ABB RobotStudio station: Solution2_20220201-115427.rsstn

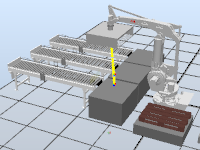
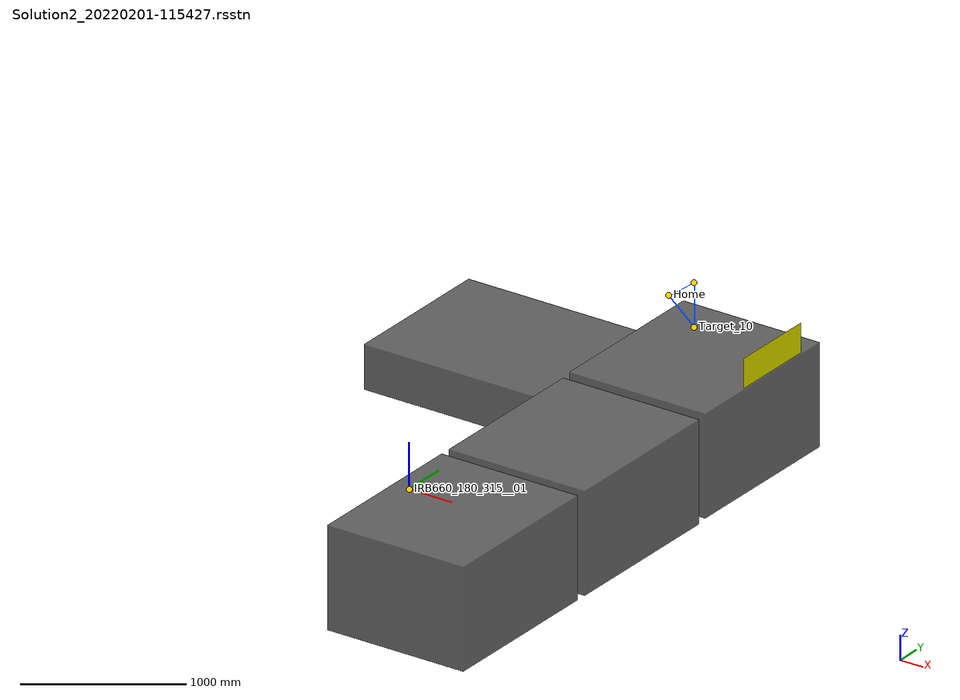
[picture v1: parts stored in the station drawn from their meshes, with robot base, taught points and paths (robot models come from the ABB library and are not in the file)]
Station Solution2 (saved by RobotStudio 21.4.9700.0)
Controller IRB660_180_315
  mechanical unit ROB_1: IRB660_180_315__01, 6 joints, base frame (0, 0, 0) mm
Layout (positions relative to the parent item):
  - IRB660_180_315__01 [mechanism, from Robots\IRB660_180_315__01.rslib] at (0, 0, 0) mm; joint values [0, 0.0198, -0.194, 0] (rad or m)
  - 600_guide [part, from Equipment\Conveyor Guide 600.rslib] at (4720, 275, 0) mm, rotated rx 0 ry 0 rz 180 deg
  - 600_guide_2 [part, from Equipment\Conveyor Guide 600.rslib] at (4720, 1475, 0) mm, rotated rx 0 ry 0 rz 180 deg
  - 600_guide_3 [part, from Equipment\Conveyor Guide 600.rslib] at (4720, -900, 0) mm, rotated rx 0 ry 0 rz 180 deg
  - 1200_4000_h2_2 [part, from Equipment\Conveyor 1200 4000 h2.rslib] at (-1500, -1000, 0) mm, rotated rx 0 ry 0 rz 180 deg
  - 1200_4000_h2_3 [part, from Equipment\Conveyor 1200 4000 h2.rslib] at (-1500, 2000, 0) mm, rotated rx 0 ry 0 rz 180 deg
  - 1200_4000_h2_4 [part, from Equipment\Conveyor 1200 4000 h2.rslib] at (-1500, 500, 0) mm, rotated rx 0 ry 0 rz 180 deg
  - 1200_4800_h2_2 [part, from Equipment\Conveyor 1200 4800 h2.rslib] at (-6865.5, 2181.45, 0) mm, rotated rx 0 ry 0 rz -90 deg
  - Pieza_1 [part] at (-5740.3, -4363.37, 0) mm, rotated rx 0 ry 0 rz 90 deg, size 1600 x 1000 x 355 mm
  - wraping_1 [part] at (-6239.59, -3461.03, 366.67) mm, rotated rx 0 ry 0 rz -90 deg, size 2370 x 1393.7 x 2100 mm
  - wraping_2 [part] at (-6238.99, -3463.39, 358.4) mm, rotated rx 0 ry 0 rz -90 deg, size 1400 x 1393.6 x 350 mm
  - wraping_3 [part] at (-6242.7, -3445.47, -111.4) mm, rotated rx 90 ry 0 rz -90 deg, size 323.7 x 500 x 658.2 mm
  - Pieza_4 [part] at (-1012.61, 969.79, 0) mm, size 1300 x 1100 x 300 mm
  - Pieza_6 [part] at (689.01, 695.64, 0) mm, size 1000 x 1200 x 700 mm
  - Pieza_7 [part] at (702.6, -1863.75, 0) mm, size 1000 x 1200 x 700 mm
  - Pieza_8 [part] at (703.57, -589.74, 0) mm, size 1000 x 1200 x 700 mm
  - Mi_mecanismo [mechanism] at (1910, 0, 2093) mm; joint values [0, 0] (rad or m)
      TCP Mi_mecanismo_1 at (1.05, 425.12, 399.16) mm, rotated rx 90 ry 0 rz 180 deg
      links: L1, L2, L3
  - Euro Pallet [graphiccomponentgroup, from Equipment\Euro Pallet.rslib] at (223.77, 1878.53, 297.19) mm, rotated rx 0 ry 0 rz 180 deg
    - Body 1 [part, from Equipment\Euro Pallet.rslib]
  - Euro Pallet_2 [graphiccomponentgroup, from Equipment\Euro Pallet.rslib] at (-1565.85, 804.31, 434.35) mm, rotated rx 0 ry 0 rz 90 deg
    - Body 1 [part, from Equipment\Euro Pallet.rslib]
  - Pieza_19 [part] at (1001.17, 2703.27, 775) mm, rotated rx 0 ry 0 rz 90 deg, size 425 x 325 x 180 mm
  - Componente inteligente_1 [smart component]
      signals: DI Start, DI Cinta, DI Coger, DI Soltar, DO Sensor1
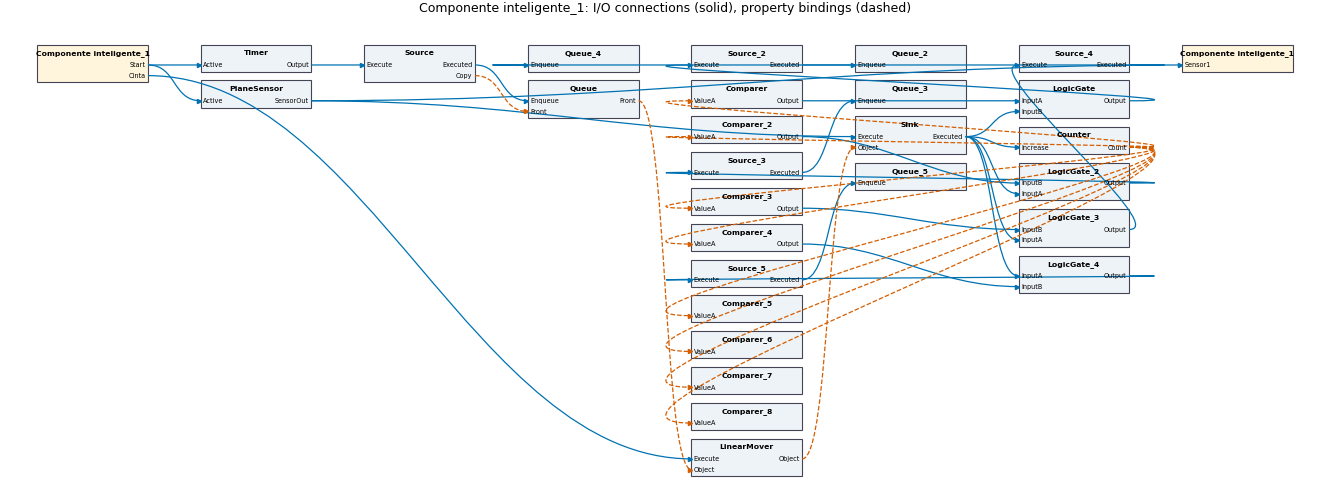
      connections:
        Componente inteligente_1.Start -> Timer.Active
        Timer.Output -> Source.Execute
        Source.Executed -> Queue.Enqueue
        Componente inteligente_1.Cinta -> LinearMover.Execute
        Componente inteligente_1.Start -> PlaneSensor.Active
        PlaneSensor.SensorOut -> Sink.Execute
        Source_2.Executed -> Queue_2.Enqueue
        Sink.Executed -> Counter.Increase
        LogicGate.Output -> Source_2.Execute
        Comparer.Output -> LogicGate.InputA
        Sink.Executed -> LogicGate.InputB
        Comparer_2.Output -> LogicGate_2.InputB
        Sink.Executed -> LogicGate_2.InputA
        LogicGate_2.Output -> Source_3.Execute
        Source_3.Executed -> Queue_3.Enqueue
        PlaneSensor.SensorOut -> Componente inteligente_1.Sensor1
        Comparer_3.Output -> LogicGate_3.InputB
        LogicGate_3.Output -> Source_4.Execute
        Sink.Executed -> LogicGate_3.InputA
        Source_4.Executed -> Queue_4.Enqueue
        Sink.Executed -> LogicGate_4.InputA
        Comparer_4.Output -> LogicGate_4.InputB
        LogicGate_4.Output -> Source_5.Execute
        Source_5.Executed -> Queue_5.Enqueue
        Source.Copy => Queue.Front
        Queue.Front => LinearMover.Object
        LinearMover.Object => Sink.Object
        Counter.Count => Comparer.ValueA
        Counter.Count => Comparer_2.ValueA
        Counter.Count => Comparer_3.ValueA
        Counter.Count => Comparer_4.ValueA
        Counter.Count => Comparer_5.ValueA
        Counter.Count => Comparer_6.ValueA
        Counter.Count => Comparer_7.ValueA
        Counter.Count => Comparer_8.ValueA
    - LinearMover [smart component, from Components\LinearMover.rslib]
        properties: Object=(none); Direction=[-0.001 0 0]; Speed=0.7; Reference=Global; ReferenceObject=(none)
    - PlaneSensor [smart component, from Components\PlaneSensor.rslib] at (1831.92, 892.97, 831.06) mm, rotated rx 0 ry -90 rz 0 deg
        properties: Origin=[0 0 0]; Axis1=[0.2 0 0]; Axis2=[0 0.6 0]; SensedPart=(none)
      - _sensorPart_ [part], size 200 x 600 x 0 mm
    - Attacher [smart component, from Components\Attacher.rslib]
        properties: Parent=(none); Flange=0; Child=(none); Mount=false; Offset=[0 0 0]; Orientation=[0 0 0]
    - Detacher [smart component, from Components\Detacher.rslib]
        properties: Child=(none); KeepPosition=true
    - Queue [smart component, from Components\Queue.rslib]
        properties: Back=(none); Front=(none); Queue=; NumberOfObjects=0
    - Source [smart component, from Components\Source.rslib]
        properties: Source=Pieza_19; Copy=(none); Parent=(none); Position=[4.6 0.975 0.775]; Orientation=[0 0 1.5707963267949]; Transient=true; PhysicsBehavior=0
    - Timer [smart component, from Components\Timer.rslib]
        properties: StartTime=0; Interval=4; Repeat=true; CurrentTime=27.336
    - Sink [smart component, from Components\Sink.rslib]
        properties: Object=(none)
    - Source_2 [smart component, from Components\Source.rslib]
        properties: Source=Pieza_19; Copy=(none); Parent=(none); Position=[1.015 1.47 0.7]; Orientation=[0 0 1.5707963267949]; Transient=false; PhysicsBehavior=0
    - Source_3 [smart component, from Components\Source.rslib]
        properties: Source=Pieza_19; Copy=(none); Parent=(none); Position=[1.345 1.47 0.7]; Orientation=[0 0 1.5707963267949]; Transient=false; PhysicsBehavior=0
    - Source_4 [smart component, from Components\Source.rslib]
        properties: Source=Pieza_19; Copy=(none); Parent=(none); Position=[1.675 1.47 0.7]; Orientation=[0 0 1.5707963267949]; Transient=false; PhysicsBehavior=0
    - Queue_2 [smart component, from Components\Queue.rslib]
        properties: Back=(none); Front=(none); Queue=; NumberOfObjects=0
    - Counter [smart component, from Components\Counter.rslib]
        properties: Count=5
    - LogicGate [smart component, from Components\LogicGate.rslib]
        properties: Operator=AND; Delay=0
    - Comparer [smart component, from Components\Comparer.rslib]
        properties: ValueA=5; Operator===; ValueB=1
    - Comparer_2 [smart component, from Components\Comparer.rslib]
        properties: ValueA=5; Operator===; ValueB=2
    - Comparer_3 [smart component, from Components\Comparer.rslib]
        properties: ValueA=5; Operator===; ValueB=3
    - Comparer_4 [smart component, from Components\Comparer.rslib]
        properties: ValueA=5; Operator===; ValueB=4
    - Comparer_5 [smart component, from Components\Comparer.rslib]
        properties: ValueA=5; Operator===; ValueB=0
    - Comparer_6 [smart component, from Components\Comparer.rslib]
        properties: ValueA=5; Operator===; ValueB=0
    - Comparer_7 [smart component, from Components\Comparer.rslib]
        properties: ValueA=5; Operator===; ValueB=0
    - LogicGate_2 [smart component, from Components\LogicGate.rslib]
        properties: Operator=AND; Delay=0
    - LogicGate_3 [smart component, from Components\LogicGate.rslib]
        properties: Operator=AND; Delay=0
    - LogicGate_4 [smart component, from Components\LogicGate.rslib]
        properties: Operator=AND; Delay=0
    - LogicGate_5 [smart component, from Components\LogicGate.rslib]
        properties: Operator=AND; Delay=0
    - LogicGate_6 [smart component, from Components\LogicGate.rslib]
        properties: Operator=AND; Delay=0
    - LogicGate_7 [smart component, from Components\LogicGate.rslib]
        properties: Operator=AND; Delay=0
    - Queue_3 [smart component, from Components\Queue.rslib]
        properties: Back=(none); Front=(none); Queue=; NumberOfObjects=0
    - Queue_4 [smart component, from Components\Queue.rslib]
        properties: Back=(none); Front=(none); Queue=; NumberOfObjects=0
    - Queue_5 [smart component, from Components\Queue.rslib]
        properties: Back=(none); Front=(none); Queue=; NumberOfObjects=0
    - Queue_6 [smart component, from Components\Queue.rslib]
        properties: Back=(none); Front=(none); Queue=; NumberOfObjects=0
    - Queue_7 [smart component, from Components\Queue.rslib]
        properties: Back=(none); Front=(none); Queue=; NumberOfObjects=0
    - Queue_8 [smart component, from Components\Queue.rslib]
        properties: Back=(none); Front=(none); Queue=; NumberOfObjects=0
    - Source_5 [smart component, from Components\Source.rslib]
        properties: Source=Pieza_19; Copy=(none); Parent=(none); Position=[0.675 1.14 0.7]; Orientation=[0 0 0]; Transient=false; PhysicsBehavior=0
    - Source_6 [smart component, from Components\Source.rslib]
        properties: Source=(none); Copy=(none); Parent=(none); Position=[0 0 0]; Orientation=[0 0 0]; Transient=false; PhysicsBehavior=0
    - Source_7 [smart component, from Components\Source.rslib]
        properties: Source=(none); Copy=(none); Parent=(none); Position=[0 0 0]; Orientation=[0 0 0]; Transient=false; PhysicsBehavior=0
    - Source_8 [smart component, from Components\Source.rslib]
        properties: Source=(none); Copy=(none); Parent=(none); Position=[0 0 0]; Orientation=[0 0 0]; Transient=false; PhysicsBehavior=0
    - Comparer_8 [smart component, from Components\Comparer.rslib]
        properties: ValueA=5; Operator===; ValueB=0
Attachment: Mi_mecanismo is attached to IRB660_180_315__01 / Link6
Attachment: PlaneSensor is attached to 1200_4800_h2_2
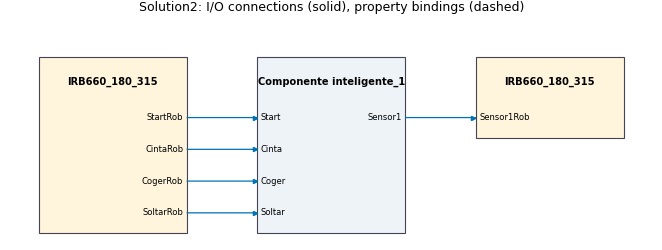
Station logic (signal -> signal, property => property):
  IRB660_180_315.StartRob -> Componente inteligente_1.Start
  IRB660_180_315.CintaRob -> Componente inteligente_1.Cinta
  IRB660_180_315.CogerRob -> Componente inteligente_1.Coger
  IRB660_180_315.SoltarRob -> Componente inteligente_1.Soltar
  Componente inteligente_1.Sensor1 -> IRB660_180_315.Sensor1Rob
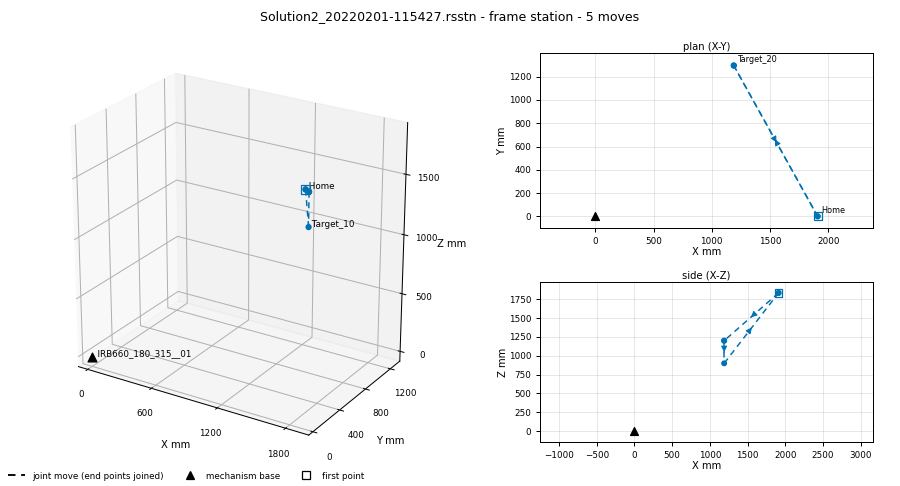
[picture p0: tool path of Solution2_20220201-115427.rsstn in frame station, 5 of 5 moves have a stored position in this frame; points joined in program order, loops and branches not executed]
Targets, tools, work objects and paths stored in the station, written as RAPID:
! task T_ROB1
MODULE CalibData
  TASK PERS wobjdata pequeño:=[FALSE,TRUE,"",[[0,0,0],[1,0,0,0]],[[0,0,0],[1,0,0,0]]];
  TASK PERS wobjdata Mediano:=[FALSE,TRUE,"",[[0,0,0],[1,0,0,0]],[[0,0,0],[1,0,0,0]]];
  TASK PERS wobjdata Grande:=[FALSE,TRUE,"",[[0,0,0],[1,0,0,0]],[[0,0,0],[1,0,0,0]]];
  PERS tooldata Servo:=[TRUE,[[0,0,114.2],[1,0,0,0]],[0.215,[8.7,12.3,49.2],[1,0,0,0],0.00021,0.00024,0.00009]];
  PERS tooldata Gripper:=[TRUE,[[0,-0.226,3866.059],[1,0,0,0]],[60,[0,0,200],[1,0,0,0],0,0,0]];
  PERS tooldata Mi_mecanismo_1:=[TRUE,[[0,0,260],[1,0,0,0]],[60,[0,0,-280],[1,0,0,0],0,0,0]];
ENDMODULE

! task T_ROB1
MODULE Module1
  CONST robtarget Home:=[[1909.999941719,0,1832.999945473],[0,0,1,0],[0,0,0,0],[9E+09,9E+09,9E+09,9E+09,9E+09,9E+09]];
  CONST robtarget Target_10:=[[1189.01,1295.635,900],[0,0,1,0],[0,0,0,0],[9E+09,9E+09,9E+09,9E+09,9E+09,9E+09]];
  CONST robtarget Target_20:=[[1189.01,1295.635,1200],[0,0,1,0],[0,0,0,0],[9E+09,9E+09,9E+09,9E+09,9E+09,9E+09]];
  PROC Path_10()
    MoveJ Home,v1000,fine,Mi_mecanismo_1\WObj:=wobj0;
    MoveJ Target_20,v1000,fine,Mi_mecanismo_1\WObj:=wobj0;
    MoveJ Target_20,v1000,fine,Mi_mecanismo_1\WObj:=wobj0;
    MoveJ Target_10,v1000,fine,Mi_mecanismo_1\WObj:=wobj0;
    MoveJ Home,v1000,fine,Mi_mecanismo_1\WObj:=wobj0;
  ENDPROC
  PROC main()
    SetDO CogerRob,0;
    SetDO SoltarRob,0;
    SetDO StartRob,1;
    SetDO CintaRob,1;
    SetDO CintaRob,0;
  ENDPROC
ENDMODULE

! task T_ROB1
MODULE pmrcUser
  TASK PERS wobjdata pmInfeeder1_WObj:=[FALSE,TRUE,"",[[0,0,0],[1,0,0,0]],[[0,0,0],[1,0,0,0]]];
  TASK PERS wobjdata pmInfeeder2_WObj:=[FALSE,TRUE,"",[[0,0,0],[1,0,0,0]],[[0,0,0],[1,0,0,0]]];
  TASK PERS wobjdata pmInfeeder3_WObj:=[FALSE,TRUE,"",[[0,0,0],[1,0,0,0]],[[0,0,0],[1,0,0,0]]];
  TASK PERS wobjdata pmInfeeder4_WObj:=[FALSE,TRUE,"",[[0,0,0],[1,0,0,0]],[[0,0,0],[1,0,0,0]]];
  TASK PERS wobjdata pmOutfeeder1_WObj:=[FALSE,TRUE,"",[[0,0,0],[1,0,0,0]],[[0,0,0],[1,0,0,0]]];
  TASK PERS wobjdata pmOutfeeder2_WObj:=[FALSE,TRUE,"",[[0,0,0],[1,0,0,0]],[[0,0,0],[1,0,0,0]]];
  TASK PERS wobjdata pmOutfeeder3_WObj:=[FALSE,TRUE,"",[[0,0,0],[1,0,0,0]],[[0,0,0],[1,0,0,0]]];
  TASK PERS wobjdata pmOutfeeder4_WObj:=[FALSE,TRUE,"",[[0,0,0],[1,0,0,0]],[[0,0,0],[1,0,0,0]]];
  TASK PERS wobjdata pmPallet1_WObj:=[FALSE,TRUE,"",[[0,0,0],[1,0,0,0]],[[0,0,0],[1,0,0,0]]];
  TASK PERS wobjdata pmSlipsheet1_WObj:=[FALSE,TRUE,"",[[0,0,0],[1,0,0,0]],[[0,0,0],[1,0,0,0]]];
  TASK PERS tooldata pmPickTool1:=[TRUE,[[0,0,0],[1,0,0,0]],[0.001,[0,0,0.001],[1,0,0,0],0,0,0]];
  TASK PERS tooldata pmSearchTool1:=[TRUE,[[0,0,0],[1,0,0,0]],[0.001,[0,0,0.001],[1,0,0,0],0,0,0]];
  TASK PERS tooldata pmCalibTool1:=[TRUE,[[0,0,0],[1,0,0,0]],[0.001,[0,0,0.001],[1,0,0,0],0,0,0]];
  PROC PmLoadReadySignalReset()
    SetDO pmSystem_doLoadReady1,0;
    SetDO pmSystem_doLoadReady2,0;
    SetDO pmSystem_doLoadReady3,0;
    SetDO pmSystem_doLoadReady4,0;
    SetDO pmSystem_doLoadReady5,0;
    SetDO pmSystem_doLoadReady6,0;
  ENDPROC
  PROC PmLoadReady()
    SetDO \Sync,pmSystem_doLoadReady1,1;
    SetDO \Sync,pmSystem_doLoadReady2,1;
    SetDO \Sync,pmSystem_doLoadReady3,1;
    SetDO \Sync,pmSystem_doLoadReady4,1;
    SetDO \Sync,pmSystem_doLoadReady5,1;
    SetDO \Sync,pmSystem_doLoadReady6,1;
  ENDPROC
  PROC PmResetProjStartFlagAtStart()
  ENDPROC
ENDMODULE

! task T_ROB1
MODULE pmrcSys
  TASK PERS wobjdata pm_home_WObj:=[FALSE,TRUE,"",[[0,0,0],[1,0,0,0]],[[0,0,0],[1,0,0,0]]];
  LOCAL PERS tooldata curr_Tool:=[TRUE,[[0,0,0],[1,0,0,0]],[0.001,[0,0,0.001],[1,0,0,0],0,0,0]];
  TASK PERS tooldata PmLastTool:=[TRUE,[[0,0,0],[1,0,0,0]],[0.001,[0,0,0.001],[1,0,0,0],0,0,0]];
  LOCAL PERS wobjdata curr_WObj:=[FALSE,TRUE,"",[[0,0,0],[1,0,0,0]],[[0,0,0],[1,0,0,0]]];
  TASK PERS wobjdata PmLastWobj:=[FALSE,TRUE,"",[[0,0,0],[1,0,0,0]],[[0,0,0],[1,0,0,0]]];
  PROC PmSetupDummyIO()
  ENDPROC
ENDMODULE

